(* IEC 61131-3 sources: SIGMATEK-Jumag-Utils-Examples/math/Class/trunc, 1 file *)

(* ---- trunc.st ---- *)
(*!
<Class
	Name               = "trunc"
	Revision           = "0.0"
	RealtimeTask       = "false"
	CyclicTask         = "true"
	BackgroundTask     = "false"
	Sigmatek           = "false"
	OSInterface        = "false"
	HighPriority       = "false"
	Automatic          = "false"
	UpdateMode         = "Prescan"
	SharedCommandTable = "true"
	Objectsize         = "(570,360)">
	<Channels>
		<Server Name="ClassSvr" Visualized="false" Initialize="false" WriteProtected="true" Retentive="false"/>
		<Server Name="DecimalPoint_0" Visualized="false" Initialize="false" WriteProtected="true" Retentive="false"/>
		<Server Name="DecimalPoint_1" Visualized="false" Initialize="false" WriteProtected="true" Retentive="false"/>
		<Server Name="DecimalPoint_2" Visualized="false" Initialize="false" WriteProtected="true" Retentive="false"/>
		<Server Name="raw" Visualized="false" Initialize="true" DefValue="125.678906" WriteProtected="false" Retentive="false"/>
	</Channels>
	<Dependencies>
		<Files>
			<File Path=".\Source\math.c"/>
		</Files>
	</Dependencies>
</Class>
*)
trunc : CLASS
  //Servers:
	ClassSvr 	: SvrChCmd_DINT;
	raw 	: SvrCh_DINT;
	DecimalPoint_0 	: SvrCh_DINT;
	DecimalPoint_1 	: SvrCh_DINT;
	DecimalPoint_2 	: SvrCh_DINT;
  //Clients:
  //Variables:
  //Functions:

	FUNCTION VIRTUAL GLOBAL CyWork
		VAR_INPUT
			EAX 	: UDINT;
		END_VAR
		VAR_OUTPUT
			state (EAX) 	: UDINT;
		END_VAR;
  //Tables:
	FUNCTION @STD
		VAR_OUTPUT
			ret_code	: CONFSTATES;
		END_VAR;
	FUNCTION GLOBAL TAB @CT_;
END_CLASS;

Function Global __cdecl truncate
VAR_INPUT
  INPUT : DINT;
  BASE : DINT;
  DIGITS : DINT;
END_VAR
VAR_OUTPUT
  Q : DINT;
END_VAR;

FUNCTION VIRTUAL GLOBAL trunc::CyWork
	VAR_INPUT
		EAX 	: UDINT;
	END_VAR
	VAR_OUTPUT
		state (EAX) 	: UDINT;
	END_VAR

  DecimalPoint_0 := truncate(INPUT:=raw, BASE:=10, DIGITS:=0);;
  DecimalPoint_1 := truncate(INPUT:=raw, BASE:=10, DIGITS:=1);;
  DecimalPoint_2 := truncate(INPUT:=raw, BASE:=10, DIGITS:=2);;

	state := READY;

END_FUNCTION
